// TIA Portal V20 export
TYPE "zp_CITITradeCalls"
// stored: Access Published, Namespace CITI_Logic
   STRUCT
      Call_1 : Bool;
      Call_2 : Bool;
      Call_3 : Bool;
      Call_4 : Bool;
      Call_5 : Bool;
      Call_6 : Bool;
      Call_7 : Bool;
      Call_8 : Bool;
      CallAck_1 : Bool;
      CallAck_2 : Bool;
      CallAck_3 : Bool;
      CallAck_4 : Bool;
      CallAck_5 : Bool;
      CallAck_6 : Bool;
      CallAck_7 : Bool;
      CallAck_8 : Bool;
   END_STRUCT;
END_TYPE
